// TIA Portal V15.1 export
// export: Created 2020-12-23T12:53:55.1483535Z, ExportSetting WithDefaults, WithReadOnly, DisplayName Totally Integrated Automation Portal, DisplayVersion V15.1 Update 3, DisplayName TIA Portal Openness, DisplayVersion V15.1, DisplayName STEP 7 Professional, DisplayVersion V15.1 Update 3, DisplayName WinCC Advanced, DisplayVersion V15.1 Update 3
FUNCTION "func_outputs" : Void   // FC1331, LAD
TITLE = OUTPUTS
{ S7_Optimized_Access := 'TRUE' }
VERSION : 0.1
// stored: AutoNumber false, CodeModifiedDate 2020-12-23T12:53:21.0067533Z, CompileDate 2020-12-23T12:53:51.673862Z, CreationDate 2020-12-23T07:31:02.6354064Z, HandleErrorsWithinBlock false, InterfaceModifiedDate 2020-12-23T12:48:47.2749857Z, IsConsistent true, IsIECCheckEnabled false, IsKnowHowProtected false, IsWriteProtected false, LibraryConformanceStatus The object is library-conformant., ModifiedDate 2020-12-23T12:53:38.1882563Z, ParameterModified 2020-12-23T07:31:02.6354064Z, PLCSimAdvancedSupport false, SetENOAutomatically False, StructureModified 2020-12-23T07:31:02.6354064Z, UDAEnableTagReadback false
BEGIN

REGION Network 1: ======= VALVES =======
END_REGION

REGION Network 2: ======= TESTS =======
END_REGION

REGION Network 3: TEST - LAMPS
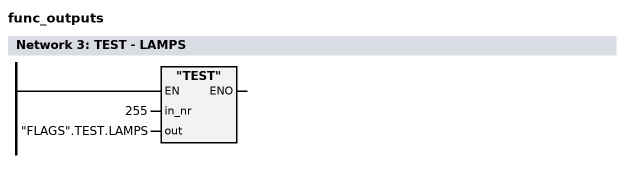
   RUNG wire#powerrail
      "TEST"(in_nr := 255, out := "FLAGS".TEST.LAMPS)
   END_RUNG
   // the same network as SCL:
   "TEST"(in_nr := 255, out := "FLAGS".TEST.LAMPS);
END_REGION
END_FUNCTION
